// TIA Portal V17 export
// export: Created 2023-03-08T16:44:23.1874801Z, ExportSetting None, DisplayName Totally Integrated Automation Portal, DisplayVersion V17 Update 4, DisplayName TIA Portal Openness, DisplayVersion V17 Update 4, DisplayName TIA Portal Version Control Interface, DisplayVersion V17, DisplayName STEP 7 Professional, DisplayVersion V17 Update 4, DisplayName STEP 7 Safety, DisplayVersion V17, DisplayName WinCC Advanced / Unified PC, DisplayVersion V17 Update 4
DATA_BLOCK "DI"   // DB12
{ S7_Optimized_Access := 'TRUE' }
// stored: AutoNumber false, MemoryReserve 100
   VAR
      KF_414 : Bool;   // DCS EMERGENCY SHUTDOWN PERSONNEL
      KF_415 : Bool;   // REMOTE FAST STOP COMPRESSOR
      TBD : Bool;   // TRIP FROM ESD
      XS_202 : Bool;   // EMERGENCY RELAY FEEDBACK
      HS_330 : Bool;   // EMERGENCY STOP PUSHBUTTON FROM UCP
      KF_403 : Bool;   // CONTROL VIA HW INTERFACE
      KF_405 : Bool;   // REMOTE START COMPRESSOR
      KF_404 : Bool;   // REMOTE STOP COMPRESSOR
      KF_406 : Bool;   // REMOTE PRODUCTION
      KF_407 : Bool;   // REMOTE RESET
      XS_100 : Bool;   // MAIN MOTOR RUNNING FEEDBACK
      XS_101 : Bool;   // MAIN MOTOR FAULT FEEDBACK
      XS_102 : Bool;   // EMERGENCY STOP FROM MCC
      XS_103 : Bool;   // HIGH TEMPERATURE FROM MCC
      XS_104 : Bool;   // MAIN CIRCUIT BREAKER FAULT
      TSH_001 : Bool;   // UCP INTERNAL HIGH TEMPERATURE
      PSA_001 : Bool;   // UCP 24VDC POWER SUPPLY FAULT
      HS_320 : Bool;   // LOCAL/REMOTE SELECTOR
      HS_340 : Bool;   // COMPRESSOR START BUTTON
      HS_350 : Bool;   // COMPRESSOR STOP BUTTON
      HS_360 : Bool;   // ALARM RESET
   END_VAR
BEGIN
END_DATA_BLOCK
